FUNCTION_BLOCK OUT_EVENT (* Event Output Flasher *)
  (* Standard: 61499-1 *)
  (* Version 0.1, 2002-05-03, JHC, Rockwell Automation, Made QI IV=true. *)
  (* Version 0.1, 2001-04-14, JHC, Rockwell Automation, Saved layout. *)
  (* Version 0.0, 2000-05-01, JHC, Rockwell Automation *)
  (* Compiler header: package fb.rt.hmi; *)
  (* Compiler Java IBM VisualAge 3.0 *)
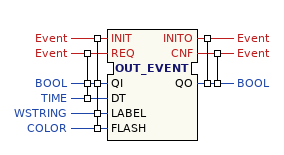
  EVENT_INPUT
    INIT WITH QI, LABEL, FLASH; (* Initialization *)
    REQ WITH QI, DT; (* Request *)
  END_EVENT
  EVENT_OUTPUT
    INITO WITH QO; (* Initialization Confirm *)
    CNF WITH QO; (* Service Confirmation *)
  END_EVENT
  VAR_INPUT
    QI : BOOL := true; (* Input event qualifier *)
    DT : TIME := t#500ms; (* Flash interval *)
    LABEL : WSTRING;
    FLASH : COLOR := COLOR#red;
  END_VAR
  VAR_OUTPUT
    QO : BOOL; (* Output event qualifier *)
  END_VAR
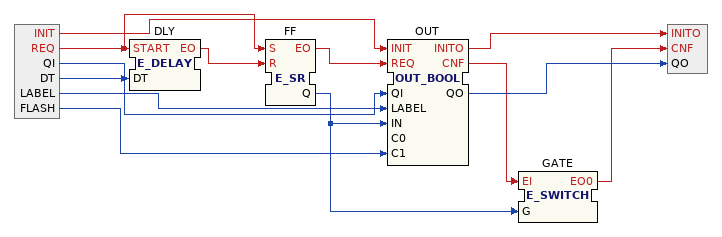
  FBS
    DLY : E_DELAY;
    FF : E_SR;
    OUT : OUT_BOOL;
    GATE : E_SWITCH;
  END_FBS
  EVENT_CONNECTIONS
    INIT TO OUT.INIT;
    OUT.INITO TO INITO;
    REQ TO DLY.START;
    REQ TO FF.S;
    DLY.EO TO FF.R;
    FF.EO TO OUT.REQ;
    OUT.CNF TO GATE.EI;
    GATE.EO0 TO CNF;
  END_CONNECTIONS
  DATA_CONNECTIONS
    QI TO OUT.QI;
    OUT.QO TO QO;
    DT TO DLY.DT;
    FF.Q TO OUT.IN;
    LABEL TO OUT.LABEL;
    FLASH TO OUT.C1;
    FF.Q TO GATE.G;
  END_CONNECTIONS
END_FUNCTION_BLOCK
